PROGRAM S1_01_Motion_04_24
VAR
	HMI_Motion: FB_HMI_Control;
	Motion: FB_Motion2way;

	tMessageOffset: UINT;
	tNumMessagesPerRow: UINT;
	
	
	MyAdvanceInterlock: BOOL;
	MyReturnInterlock: BOOL;
	
	MyAutoAdvanceCondition: BOOL;
	MyAutoReturnCondition: BOOL;
	testword: WORD;
	myAdvancePrompt: BOOL;
	myReturnPrompt: BOOL;
END_VAR

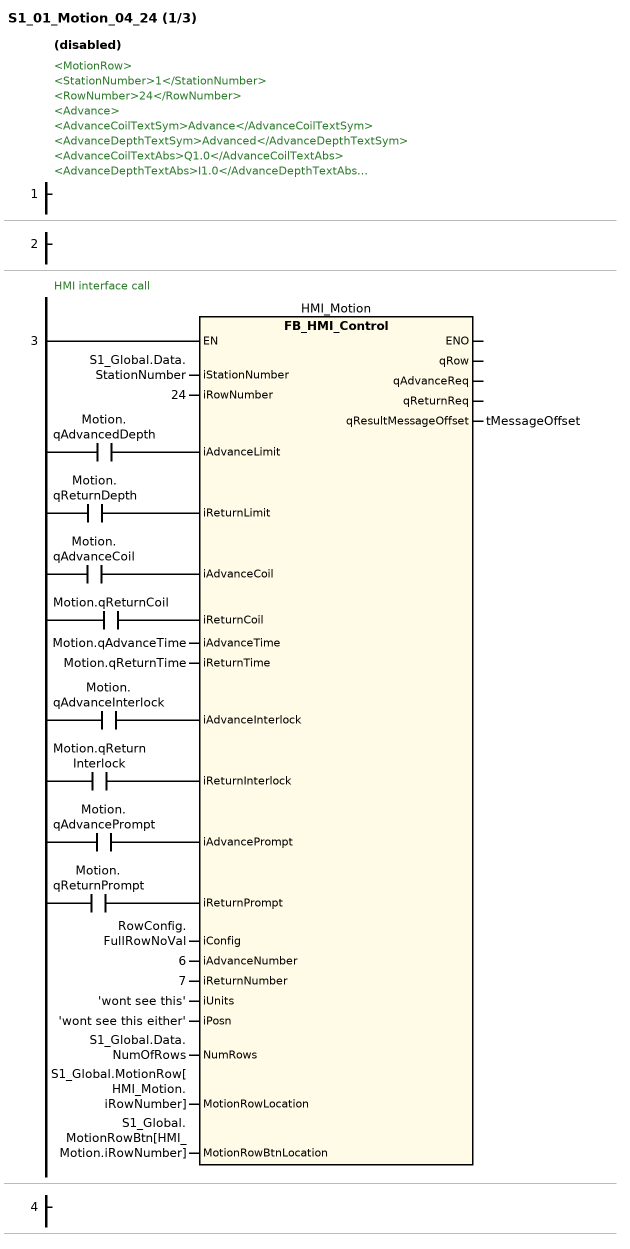
// NETWORK 1 (disabled)
// <MotionRow>
// <StationNumber>1</StationNumber>
// <RowNumber>24</RowNumber>
//   <Advance>
//     <AdvanceCoilTextSym>Advance</AdvanceCoilTextSym>
//     <AdvanceDepthTextSym>Advanced</AdvanceDepthTextSym>
//     <AdvanceCoilTextAbs>Q1.0</AdvanceCoilTextAbs>
//     <AdvanceDepthTextAbs>I1.0</AdvanceDepthTextAbs>
//     <ManSeq>1</ManSeq>
//   </Advance>
//   <Return>
//     <ReturnCoilTextSym>Return</ReturnCoilTextSym>
//     <ReturnDepthTextSym>Returned</ReturnDepthTextSym>
//     <ReturnCoilTextAbs>Q1.1</ReturnCoilTextAbs>
//     <ReturnDepthTextAbs>I1.1</ReturnDepthTextAbs>
//    <ManSeq>2</ManSeq>
//   </Return>
//   <Motion>
//     <NameSym>Clamp Cylinder</NameSym>
//     <NameAbs>A1</NameAbs>
//   </Motion>
// </MotionRow>

// NETWORK 2

// NETWORK 3
// HMI interface call
HMI_Motion(
    iStationNumber := S1_Global.Data.StationNumber,
    iRowNumber := 24,
    iAdvanceLimit := Motion.qAdvancedDepth,
    iReturnLimit := Motion.qReturnDepth,
    iAdvanceCoil := Motion.qAdvanceCoil,
    iReturnCoil := Motion.qReturnCoil,
    iAdvanceTime := Motion.qAdvanceTime,
    iReturnTime := Motion.qReturnTime,
    iAdvanceInterlock := Motion.qAdvanceInterlock,
    iReturnInterlock := Motion.qReturnInterlock,
    iAdvancePrompt := Motion.qAdvancePrompt,
    iReturnPrompt := Motion.qReturnPrompt,
    iConfig := RowConfig.FullRowNoVal,
    iAdvanceNumber := 6,
    iReturnNumber := 7,
    iUnits := 'wont see this',
    iPosn := 'wont see this either',
    NumRows := S1_Global.Data.NumOfRows,
    MotionRowLocation := S1_Global.MotionRow[HMI_Motion.iRowNumber],
    MotionRowBtnLocation := S1_Global.MotionRowBtn[HMI_Motion.iRowNumber],
    qResultMessageOffset => tMessageOffset); // FB_HMI_Control

// NETWORK 4

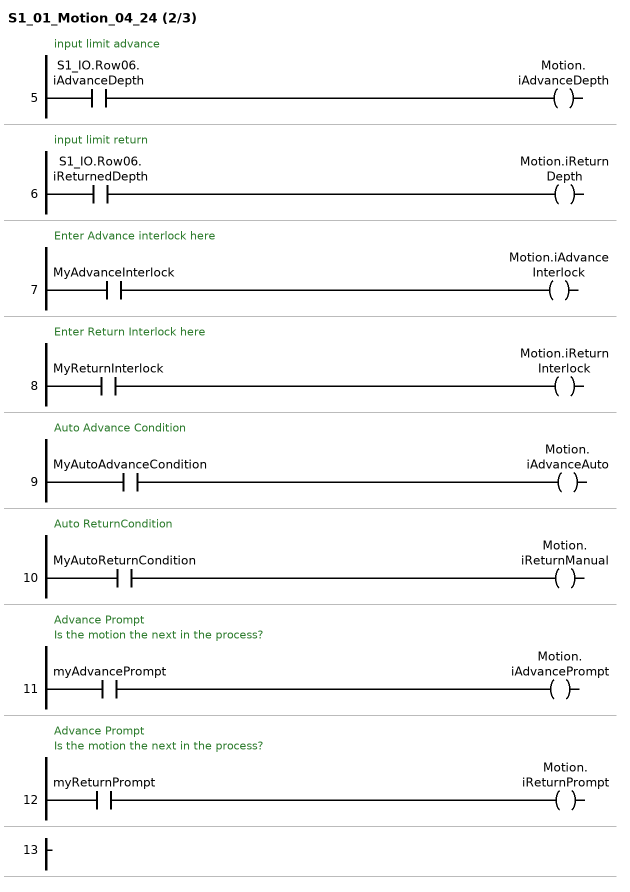
// NETWORK 5
// input limit advance
Motion.iAdvanceDepth := S1_IO.Row06.iAdvanceDepth;

// NETWORK 6
// input limit return
Motion.iReturnDepth := S1_IO.Row06.iReturnedDepth;

// NETWORK 7
// Enter Advance interlock here
Motion.iAdvanceInterlock := MyAdvanceInterlock;

// NETWORK 8
// Enter Return Interlock here
Motion.iReturnInterlock := MyReturnInterlock;

// NETWORK 9
// Auto Advance Condition
Motion.iAdvanceAuto := MyAutoAdvanceCondition;

// NETWORK 10
// Auto ReturnCondition
Motion.iReturnManual := MyAutoReturnCondition;

// NETWORK 11
// Advance Prompt
// Is the motion the next in the process?
Motion.iAdvancePrompt := myAdvancePrompt;

// NETWORK 12
// Advance Prompt
// Is the motion the next in the process?
Motion.iReturnPrompt := myReturnPrompt;

// NETWORK 13

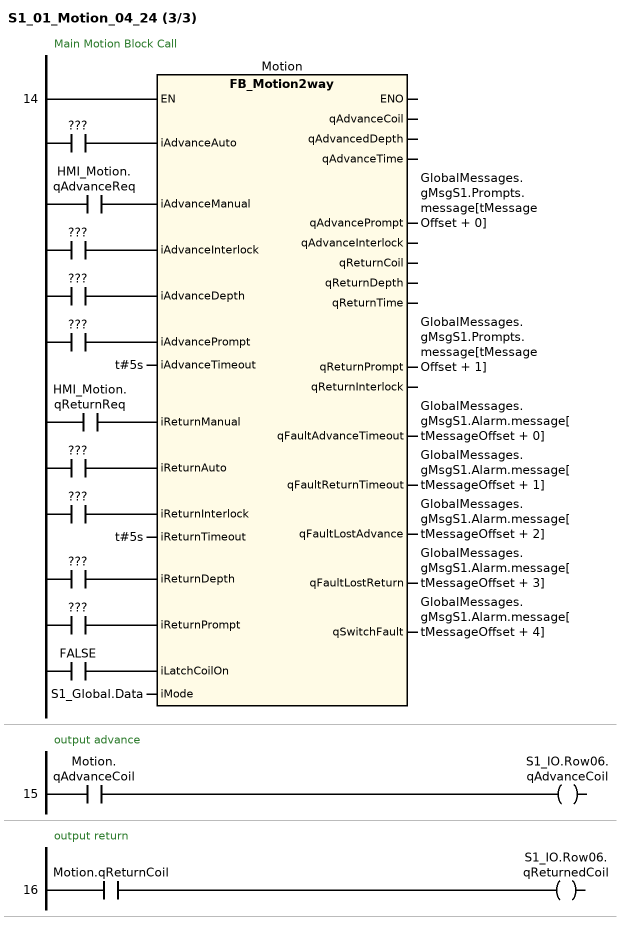
// NETWORK 14
// Main Motion Block Call
Motion(
    iAdvanceManual := HMI_Motion.qAdvanceReq,
    iAdvanceTimeout := t#5s,
    iReturnManual := HMI_Motion.qReturnReq,
    iReturnTimeout := t#5s,
    iLatchCoilOn := FALSE,
    iMode := S1_Global.Data,
    qAdvancePrompt => GlobalMessages.gMsgS1.Prompts.message[tMessageOffset + 0],
    qReturnPrompt => GlobalMessages.gMsgS1.Prompts.message[tMessageOffset + 1],
    qFaultAdvanceTimeout => GlobalMessages.gMsgS1.Alarm.message[tMessageOffset + 0],
    qFaultReturnTimeout => GlobalMessages.gMsgS1.Alarm.message[tMessageOffset + 1],
    qFaultLostAdvance => GlobalMessages.gMsgS1.Alarm.message[tMessageOffset + 2],
    qFaultLostReturn => GlobalMessages.gMsgS1.Alarm.message[tMessageOffset + 3],
    qSwitchFault => GlobalMessages.gMsgS1.Alarm.message[tMessageOffset + 4]); // FB_Motion2way

// NETWORK 15
// output advance
S1_IO.Row06.qAdvanceCoil := Motion.qAdvanceCoil;

// NETWORK 16
// output return
S1_IO.Row06.qReturnedCoil := Motion.qReturnCoil;

END_PROGRAM

(* stored: Version 1.1.0.1, ProductVersion 3.1.4024.12
   POU S1_01_Motion_04_24: Id {31154a7b-0aec-492b-8651-7095c5499f53}, SpecialFunc None *)
